// TIA Portal project "Test_HTTP_PLC" (V15)

(* hardware
DEVICE "S7-1200 station_1"  S7-1200 Station
   slot 0: "Rack_0"  S7-1200 Rack  Rack  V1.0
   slot 1: "PLC_1"  CPU 1211C DC/DC/Rly  6ES7 211-1HE40-0XB0  V4.2
DEVICE "S71500/ET200MP station_1"  S7-1500 station
   slot 0: "Rail_0"  Rack  6ES7 590-1***0-0AA0
   slot 1: "PLC_2"  CPU 1516-3 PN/DP  6ES7 516-3AN01-0AB0  V2.5
      slot 3: "CPU display_1"  6ES7591-1BA00-0AA0
*)

// ===== PLC "PLC_1"  CPU 1211C DC/DC/Rly =====

VAR_GLOBAL   // PLC tag table "Default tag table"
   "jooj" AT %I0.0 : Bool;
END_VAR

DATA_BLOCK "DB_Change_Data"   // DB1
{ S7_Optimized_Access := 'TRUE' }
VERSION : 0.1
   VAR
      BTN_Send : Bool;
      BTN_Get : Bool;
      Result_Get : String := 'jooj';
      Result_Post : String;
   END_VAR
BEGIN
END_DATA_BLOCK

// folder: System blocks/Program resources

DATA_BLOCK "PLC_1_Send_DB"   // DB2
{ S7_Optimized_Access := 'TRUE' }
AUTHOR : SIMATIC
FAMILY : MC7Plus
NAME : TC_IP_v4
VERSION : 1.0
// stored: InstanceOfName TCON_IP_v4
"TCON_IP_v4"
BEGIN
   ID := 1;
   InterfaceId := 64;
   LocalPort := 2000;
   RemoteAddress.ADDR[1] := 10;
   RemoteAddress.ADDR[2] := 251;
   RemoteAddress.ADDR[3] := 16;
   RemoteAddress.ADDR[4] := 133;
   ConnectionType := 11;
END_DATA_BLOCK

DATA_BLOCK "PLC_1_Receive_DB"   // DB5
{ S7_Optimized_Access := 'TRUE' }
AUTHOR : SIMATIC
FAMILY : MC7Plus
NAME : TC_IP_v4
VERSION : 1.0
// stored: InstanceOfName TCON_IP_v4
"TCON_IP_v4"
BEGIN
   ID := 2;
   InterfaceId := 64;
   RemotePort := 2001;
   ActiveEstablished := true;
   RemoteAddress.ADDR[1] := 10;
   RemoteAddress.ADDR[2] := 251;
   RemoteAddress.ADDR[3] := 16;
   RemoteAddress.ADDR[4] := 133;
END_DATA_BLOCK

// folder: (top level)

ORGANIZATION_BLOCK "Main"   // OB1, LAD, ProgramCycle
TITLE = "Main Program Sweep (Cycle)"
{ S7_Optimized_Access := 'TRUE' }
VERSION : 0.1
   VAR_INPUT
      Initial_Call : Bool;   // Initial call of this OB
      Remanence : Bool;   // =True, if remanent data are available
   END_VAR
BEGIN

REGION Network 1
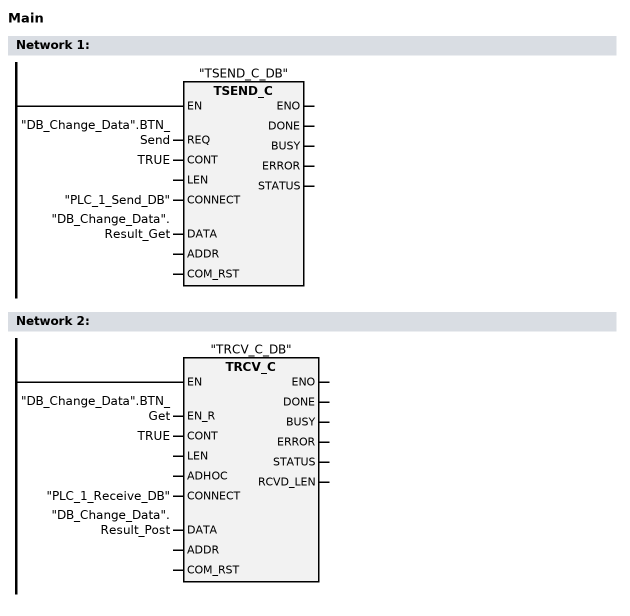
   "TSEND_C_DB"(REQ := "DB_Change_Data".BTN_Send,   // TSEND_C
                CONT := TRUE,
                CONNECT := "PLC_1_Send_DB",
                DATA := "DB_Change_Data".Result_Get);
END_REGION

REGION Network 2
   "TRCV_C_DB"(EN_R := "DB_Change_Data".BTN_Get,   // TRCV_C
               CONT := TRUE,
               CONNECT := "PLC_1_Receive_DB",
               DATA := "DB_Change_Data".Result_Post);
END_REGION
END_ORGANIZATION_BLOCK

// ===== PLC "PLC_2"  CPU 1516-3 PN/DP =====

DATA_BLOCK "DB_OPC"   // DB1
{ S7_Optimized_Access := 'FALSE' }
VERSION : 0.1
   VAR
      OPC_DATA : Struct
         Data_String : String;
         Data_Bool : Bool;
         Data_Int : Int;
      END_STRUCT;
   END_VAR
BEGIN
END_DATA_BLOCK